GLOBALCONSTANTS GlobalConstants (* Global constants *)
  (* Standard: 61499-1 *)
  (* Version 1.0, 2023-07-12, mjobst, 4DIAC-Consortium *)
END_GLOBALCONSTANTS
